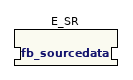
        [picture p73: application DataConnectionTestApp.Test4.nestedSubapp]
        FBS
          E_SR : fb_sourcedata;
        END_FBS
      END_SUBAPPLICATION
    END_SUBAPPLICATION
    SUBAPPLICATION Test4Solution
      EVENT_OUTPUT
        EO1;
      END_EVENT
      VAR_INPUT
        destination : BOOL;
      END_VAR
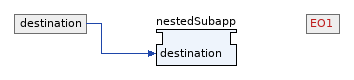
      SUBAPPLICATION nestedSubapp
        VAR_INPUT
          destination : BOOL;
        END_VAR
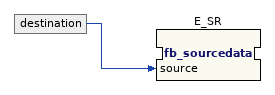
        FBS
          E_SR : fb_sourcedata;
        END_FBS
        DATA_CONNECTIONS
          destination TO E_SR.source;
        END_CONNECTIONS
      END_SUBAPPLICATION
      DATA_CONNECTIONS
        destination TO nestedSubapp.destination;
      END_CONNECTIONS
    END_SUBAPPLICATION
    SUBAPPLICATION Test5 (* crossing connection from FB to FB in nested subapp via app network *)
      EVENT_OUTPUT
        EO1;
      END_EVENT
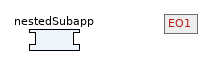
      SUBAPPLICATION nestedSubapp
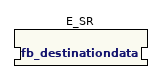
        FBS
          E_SR : fb_destinationdata;
        END_FBS
      END_SUBAPPLICATION
    END_SUBAPPLICATION
    SUBAPPLICATION Test6 (* crossing connection from FB to nested subapp interface *)
      EVENT_OUTPUT
        EO1;
      END_EVENT
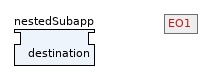
      SUBAPPLICATION nestedSubapp
        VAR_OUTPUT
          destination : BOOL;
        END_VAR
      END_SUBAPPLICATION
    END_SUBAPPLICATION
    SUBAPPLICATION Test7 (* crossing connection from FB to FB in nested subapp, one pin already exists *)
      VAR_OUTPUT
        destination : BOOL;
      END_VAR
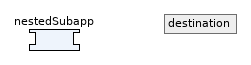
      SUBAPPLICATION nestedSubapp
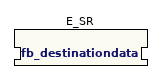
        FBS
          E_SR : fb_destinationdata;
        END_FBS
      END_SUBAPPLICATION
    END_SUBAPPLICATION
    SUBAPPLICATION Test8 (* crossing connection from FB in subapp to FB in nested subapp *)
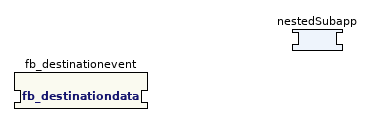
      FBS
        fb_destinationevent : fb_destinationdata;
      END_FBS
      SUBAPPLICATION nestedSubapp
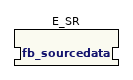
        FBS
          E_SR : fb_sourcedata;
        END_FBS
      END_SUBAPPLICATION
    END_SUBAPPLICATION
    SUBAPPLICATION Test9 (* event input pin already exists outwards *)
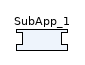
      SUBAPPLICATION SubApp_1
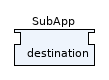
        SUBAPPLICATION SubApp
          VAR_OUTPUT
            destination : BOOL;
          END_VAR
        END_SUBAPPLICATION
      END_SUBAPPLICATION
    END_SUBAPPLICATION
    SUBAPPLICATION SubApp_8
      EVENT_INPUT
        source;
      END_EVENT
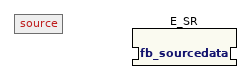
      FBS
        E_SR : fb_sourcedata;
      END_FBS
    END_SUBAPPLICATION
    SUBAPPLICATION Test10 (* event input pin with same name already exists *)
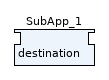
      SUBAPPLICATION SubApp_1
        VAR_INPUT
          destination : INT;
        END_VAR
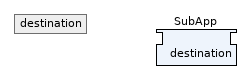
        SUBAPPLICATION SubApp
          VAR_OUTPUT
            destination : BOOL;
          END_VAR
        END_SUBAPPLICATION
      END_SUBAPPLICATION
    END_SUBAPPLICATION
    SUBAPPLICATION SubApp_10
      VAR_INPUT
        source : BOOL;
      END_VAR
    END_SUBAPPLICATION
    SUBAPPLICATION Test12 (* event input already exists inwards *)
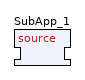
      SUBAPPLICATION SubApp_1
        EVENT_INPUT
          source;
        END_EVENT
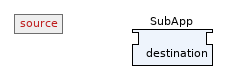
        SUBAPPLICATION SubApp
          VAR_OUTPUT
            destination : INT;
          END_VAR
        END_SUBAPPLICATION
      END_SUBAPPLICATION
    END_SUBAPPLICATION
    SUBAPPLICATION SubApp_12
      VAR_OUTPUT
        source : INT;
      END_VAR
    END_SUBAPPLICATION
    SUBAPPLICATION Test16 (* event input pin with same name already exists, inwards *)
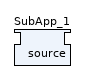
      SUBAPPLICATION SubApp_1
        VAR_OUTPUT
          source : BOOL;
        END_VAR
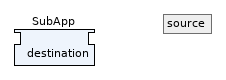
        SUBAPPLICATION SubApp
          VAR_OUTPUT
            destination : BOOL;
          END_VAR
        END_SUBAPPLICATION
      END_SUBAPPLICATION
    END_SUBAPPLICATION
    SUBAPPLICATION SubApp_14
      VAR_OUTPUT
        source : BOOL;
      END_VAR
    END_SUBAPPLICATION
    SUBAPPLICATION Test1Result (* connection between subapp borders *)
      EVENT_OUTPUT
        EO1;
      END_EVENT
      VAR_INPUT
        source : BOOL;
      END_VAR
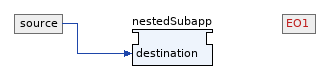
      SUBAPPLICATION nestedSubapp
        VAR_INPUT
          destination : BOOL;
        END_VAR
      END_SUBAPPLICATION
      DATA_CONNECTIONS
        source TO nestedSubapp.destination;
      END_CONNECTIONS
    END_SUBAPPLICATION
    SUBAPPLICATION Test2 (* connection between subapp borders *)
      EVENT_OUTPUT
        EO1;
      END_EVENT
      VAR_INPUT
        destination : BOOL;
      END_VAR
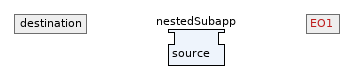
      SUBAPPLICATION nestedSubapp
        VAR_INPUT
          source : BOOL;
        END_VAR
      END_SUBAPPLICATION
    END_SUBAPPLICATION
    SUBAPPLICATION Test2Solution (* connection between subapp borders *)
      EVENT_OUTPUT
        EO1;
      END_EVENT
      VAR_INPUT
        destination : BOOL;
      END_VAR
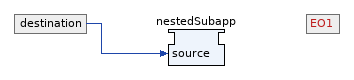
      SUBAPPLICATION nestedSubapp
        VAR_INPUT
          source : BOOL;
        END_VAR
      END_SUBAPPLICATION
      DATA_CONNECTIONS
        destination TO nestedSubapp.source;
      END_CONNECTIONS
    END_SUBAPPLICATION
    SUBAPPLICATION Test3Solution (* crossing connection from FB to subapp border *)
      EVENT_OUTPUT
        EO1;
      END_EVENT
      VAR_INPUT
        destination : BOOL;
      END_VAR
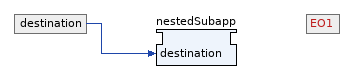
      SUBAPPLICATION nestedSubapp
        VAR_INPUT
          destination : BOOL;
        END_VAR
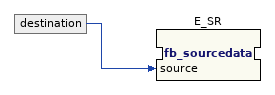
        FBS
          E_SR : fb_sourcedata;
        END_FBS
        DATA_CONNECTIONS
          destination TO E_SR.source;
        END_CONNECTIONS
      END_SUBAPPLICATION
      DATA_CONNECTIONS
        destination TO nestedSubapp.destination;
      END_CONNECTIONS
    END_SUBAPPLICATION
    SUBAPPLICATION Test5Solution (* crossing connection from FB to FB in nested subapp via app network *)
      EVENT_OUTPUT
        EO1;
      END_EVENT
      VAR_OUTPUT
        destination : BOOL;
      END_VAR
